FUNCTION_BLOCK SS5a_ps_AirNozzle (* Composite FB wrapping other FBs *)
  (* Standard: 61499-2 *)
  (* Version 1.0, 2025-08-26, PS_Transformer_for_Unknown *)
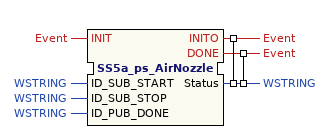
  EVENT_INPUT
    INIT; (* Initialization Request *)
  END_EVENT
  EVENT_OUTPUT
    INITO WITH Status; (* Initialization Confirm *)
    DONE WITH Status; (* Execution Confirmation *)
  END_EVENT
  VAR_INPUT
    ID_SUB_START : WSTRING;
    ID_SUB_STOP : WSTRING;
    ID_PUB_DONE : WSTRING;
  END_VAR
  VAR_OUTPUT
    Status : WSTRING; (* Output event qualifier *)
  END_VAR
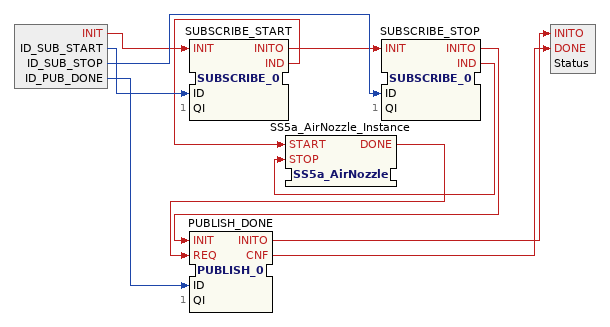
  FBS
    SS5a_AirNozzle_Instance : SS5a_AirNozzle;
    SUBSCRIBE_START : SUBSCRIBE_0(QI := 1);
    SUBSCRIBE_STOP : SUBSCRIBE_0(QI := 1);
    PUBLISH_DONE : PUBLISH_0(QI := 1);
  END_FBS
  EVENT_CONNECTIONS
    INIT TO SUBSCRIBE_START.INIT;
    SUBSCRIBE_START.INITO TO SUBSCRIBE_STOP.INIT;
    SUBSCRIBE_STOP.INITO TO PUBLISH_DONE.INIT;
    PUBLISH_DONE.INITO TO INITO;
    SUBSCRIBE_START.IND TO SS5a_AirNozzle_Instance.START;
    SUBSCRIBE_STOP.IND TO SS5a_AirNozzle_Instance.STOP;
    SS5a_AirNozzle_Instance.DONE TO PUBLISH_DONE.REQ;
    PUBLISH_DONE.CNF TO DONE;
  END_CONNECTIONS
  DATA_CONNECTIONS
    ID_SUB_START TO SUBSCRIBE_START.ID;
    ID_SUB_STOP TO SUBSCRIBE_STOP.ID;
    ID_PUB_DONE TO PUBLISH_DONE.ID;
  END_CONNECTIONS
END_FUNCTION_BLOCK
